// SIMATIC S7-200 project (STEP 7-Micro/WIN), CPU 224XP REL 02.01

SYMBOL_TABLE USUARIO1
teclado_1        I0.0
teclado_2        I0.1
teclado_3        I0.2
teclado_4        I0.3
TECLADO_ON       I0.4
teclado_5        I0.5
teclado_6        I0.6
teclado_7        I0.7
teclado_8        I1.0
teclado_9        I1.1
teclado_0        I1.2
TECLA_OFF        I1.3
PUERTA           Q0.0
LUZ              Q0.1
SIRENA           Q0.2
END_SYMBOL_TABLE

SYMBOL_TABLE Símbolos S7-200
Primer_ciclo_ON  SM0.1    // ON sólo en el primer ciclo
Reloj_1s         SM0.5    // Reloj ON durante 0,5 s, OFF durante 0,5 s, tiempo de ciclo = 1 s.
END_SYMBOL_TABLE

ORGANIZATION_BLOCK PRINCIPAL:OB1
TITLE=COMENTARIOS DEL PROGRAMA
BEGIN
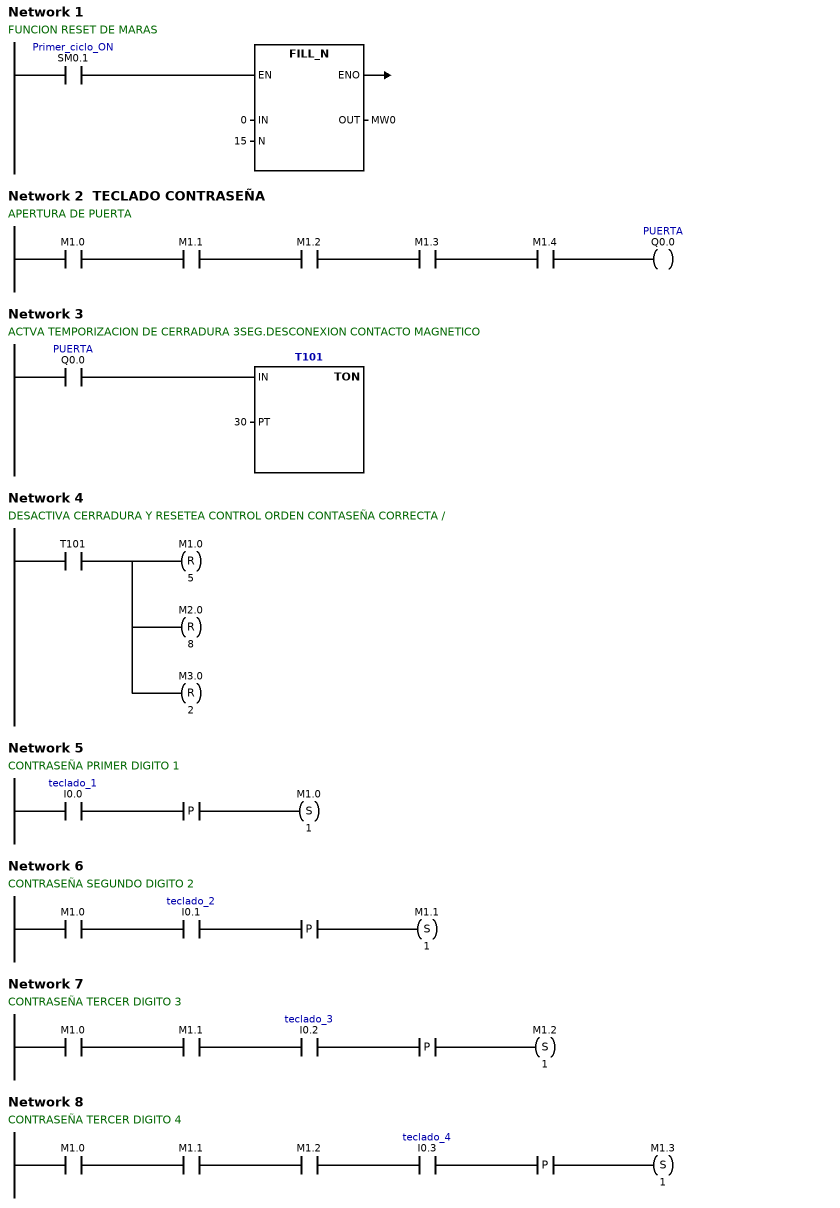
Network 1
// FUNCION RESET DE MARAS
LD     Primer_ciclo_ON:SM0.1
FILL   0, MW0, 15
Network 2 // TECLADO CONTRASEÑA
// APERTURA DE PUERTA
LD     M1.0
A      M1.1
A      M1.2
A      M1.3
A      M1.4
=      PUERTA:Q0.0
Network 3
// ACTVA TEMPORIZACION DE CERRADURA 3SEG.DESCONEXION CONTACTO MAGNETICO
LD     PUERTA:Q0.0
TON    T101, 30
Network 4
// DESACTIVA CERRADURA Y RESETEA CONTROL ORDEN CONTASEÑA CORRECTA
// 
// (network saved uncompiled; LAD cells follow)
// row 0: c0 -| |- T101 v  c1 -(R) M1.0, 5
// row 1: c0 ^v  c1 -(R) M2.0, 8
// row 2: c0 ^  c1 -(R) M3.0, 2
Network 5
// CONTRASEÑA PRIMER DIGITO 1
LD     teclado_1:I0.0
EU
S      M1.0, 1
Network 6
// CONTRASEÑA SEGUNDO DIGITO 2
LD     M1.0
A      teclado_2:I0.1
EU
S      M1.1, 1
Network 7
//  CONTRASEÑA TERCER DIGITO 3
LD     M1.0
A      M1.1
A      teclado_3:I0.2
EU
S      M1.2, 1
Network 8
// CONTRASEÑA TERCER DIGITO 4
LD     M1.0
A      M1.1
A      M1.2
A      teclado_4:I0.3
EU
S      M1.3, 1
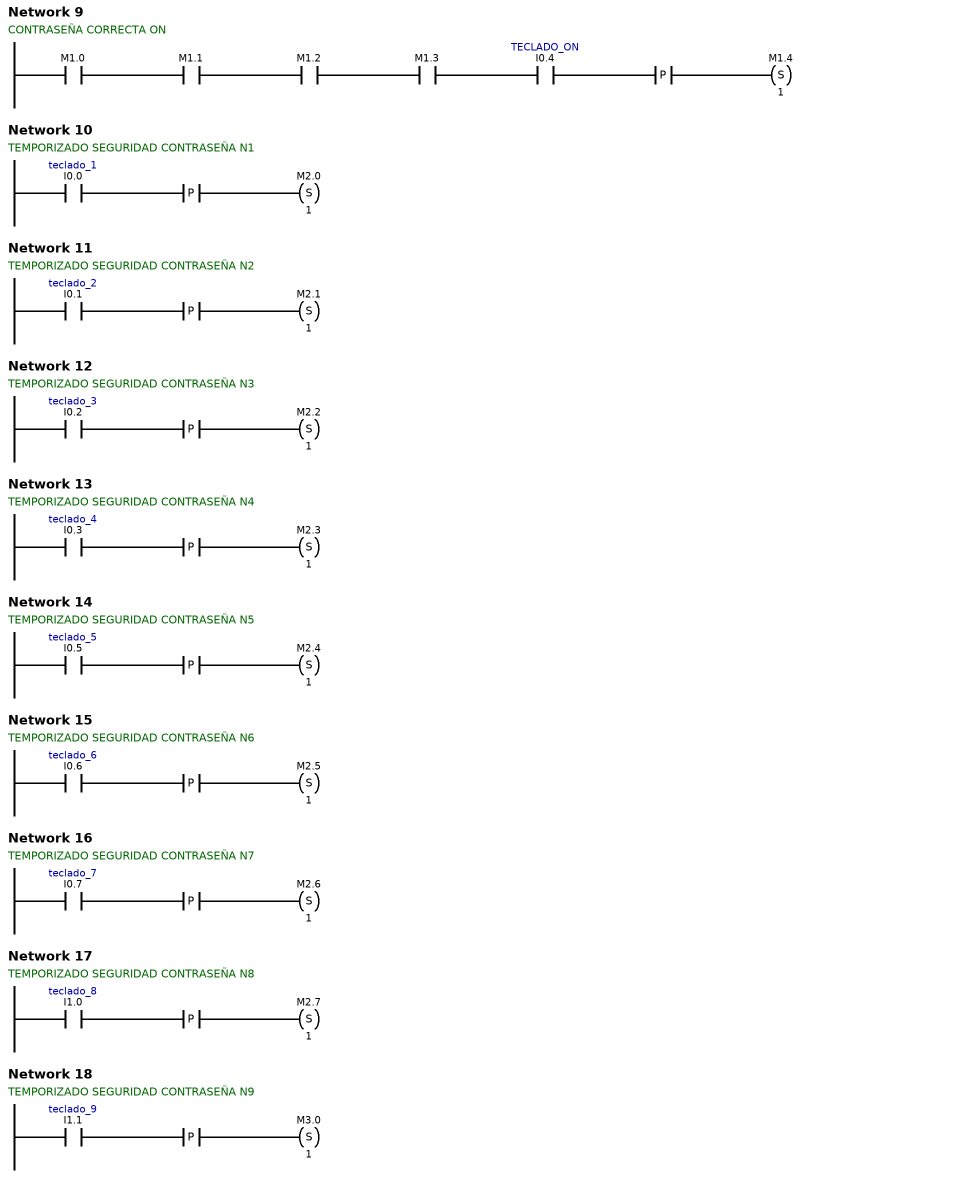
Network 9
// CONTRASEÑA CORRECTA ON
LD     M1.0
A      M1.1
A      M1.2
A      M1.3
A      TECLADO_ON:I0.4
EU
S      M1.4, 1
Network 10
// TEMPORIZADO SEGURIDAD CONTRASEÑA N1
LD     teclado_1:I0.0
EU
S      M2.0, 1
Network 11
// TEMPORIZADO SEGURIDAD CONTRASEÑA N2
LD     teclado_2:I0.1
EU
S      M2.1, 1
Network 12
// TEMPORIZADO SEGURIDAD CONTRASEÑA N3
LD     teclado_3:I0.2
EU
S      M2.2, 1
Network 13
// TEMPORIZADO SEGURIDAD CONTRASEÑA N4
LD     teclado_4:I0.3
EU
S      M2.3, 1
Network 14
// TEMPORIZADO SEGURIDAD CONTRASEÑA N5
LD     teclado_5:I0.5
EU
S      M2.4, 1
Network 15
// TEMPORIZADO SEGURIDAD CONTRASEÑA N6
LD     teclado_6:I0.6
EU
S      M2.5, 1
Network 16
// TEMPORIZADO SEGURIDAD CONTRASEÑA N7
LD     teclado_7:I0.7
EU
S      M2.6, 1
Network 17
// TEMPORIZADO SEGURIDAD CONTRASEÑA N8
LD     teclado_8:I1.0
EU
S      M2.7, 1
Network 18
// TEMPORIZADO SEGURIDAD CONTRASEÑA N9
LD     teclado_9:I1.1
EU
S      M3.0, 1
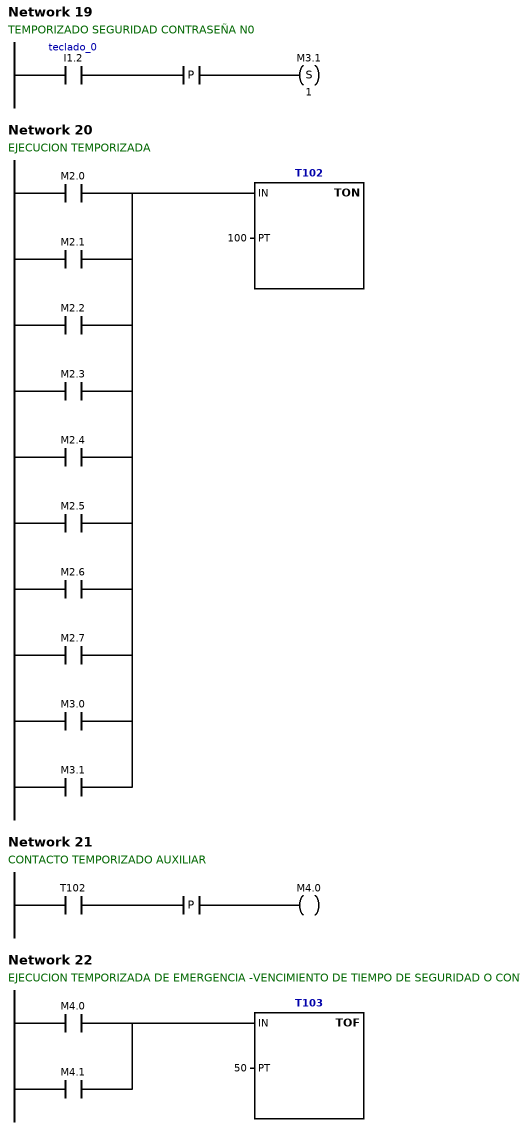
Network 19
// TEMPORIZADO SEGURIDAD CONTRASEÑA N0
LD     teclado_0:I1.2
EU
S      M3.1, 1
Network 20
// EJECUCION TEMPORIZADA 
LD     M2.0
O      M2.1
O      M2.2
O      M2.3
O      M2.4
O      M2.5
O      M2.6
O      M2.7
O      M3.0
O      M3.1
TON    T102, 100
Network 21
// CONTACTO TEMPORIZADO AUXILIAR 
LD     T102
EU
=      M4.0
Network 22
// EJECUCION TEMPORIZADA DE EMERGENCIA -VENCIMIENTO DE TIEMPO DE SEGURIDAD O CONTRASEÑA INCORRECTA
LD     M4.0
O      M4.1
TOF    T103, 50
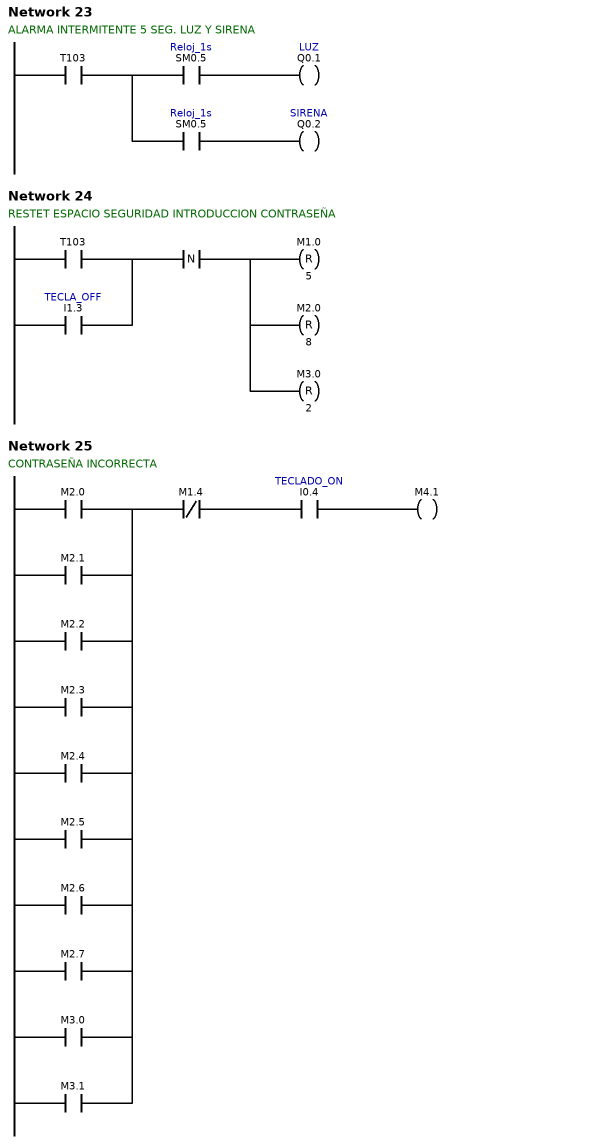
Network 23
// ALARMA INTERMITENTE 5 SEG. LUZ Y SIRENA
LD     T103
LPS
A      Reloj_1s:SM0.5
=      LUZ:Q0.1
LPP
A      Reloj_1s:SM0.5
=      SIRENA:Q0.2
Network 24
// RESTET ESPACIO SEGURIDAD INTRODUCCION CONTRASEÑA
LD     T103
O      TECLA_OFF:I1.3
ED
R      M1.0, 5
R      M2.0, 8
R      M3.0, 2
Network 25
// CONTRASEÑA INCORRECTA
LD     M2.0
O      M2.1
O      M2.2
O      M2.3
O      M2.4
O      M2.5
O      M2.6
O      M2.7
O      M3.0
O      M3.1
AN     M1.4
A      TECLADO_ON:I0.4
=      M4.1
END_ORGANIZATION_BLOCK
